{attribute 'GeneratedUsingTerminal: EP2816-0003-0016'}
{attribute addProperty BoxType "EP2816-0003-0016"}
{attribute addProperty Id "EtcSlaveTerminalBaseDIG_Diag_Inputs_Channel_1AT %I*DIG_Diag_Inputs_Channel_584303BF8DIG_Diag_Inputs_Channel_2AT %I*DIG_Diag_Inputs_Channel_584303BF8DIG_Inputs_DeviceAT %I*DIG_Inputs_Device_E94E5BF95DIG_Output_Channel_1AT %Q*DIG_Output_Channel_28AC1A9E8DIG_Output_Channel_2AT %Q*DIG_Output_Channel_28AC1A9E8DIG_Outputs_DeviceAT %Q*DIG_Outputs_Device_36A5EF172WcStateAT %I*WcState_9091E0EB2InfoDataAT %I*InfoData_32EB74EA10"}
{attribute addProperty CRC "3316017075"}
{attribute addProperty Size "51"}
TYPE EP2816_C5A667B3 EXTENDS EtcSlaveTerminalBase :
STRUCT
	{attribute addProperty Name "DIG_Diag_Inputs_Channel_1"}
	DIG_Diag_Inputs_Channel_1 : DIG_Diag_Inputs_Channel_584303BF;
	{attribute addProperty Name "DIG_Diag_Inputs_Channel_2"}
	DIG_Diag_Inputs_Channel_2 : DIG_Diag_Inputs_Channel_584303BF;
	{attribute addProperty Name "DIG_Inputs_Device"}
	DIG_Inputs_Device : DIG_Inputs_Device_E94E5BF9;
	{attribute addProperty Name "DIG_Output_Channel_1"}
	DIG_Output_Channel_1 : DIG_Output_Channel_28AC1A9E;
	{attribute addProperty Name "DIG_Output_Channel_2"}
	DIG_Output_Channel_2 : DIG_Output_Channel_28AC1A9E;
	{attribute addProperty Name "DIG_Outputs_Device"}
	DIG_Outputs_Device : DIG_Outputs_Device_36A5EF17;
	{attribute addProperty Name "WcState"}
	WcState : WcState_9091E0EB;
	{attribute addProperty Name "InfoData"}
	InfoData : InfoData_32EB74EA;
END_STRUCT
END_TYPE

(* stored: Version 1.2.0.0, ProductVersion 3.1.4024.9
   DUT EP2816_C5A667B3: Id {a648cb08-7737-4b96-b226-0bf649375767} *)
